// TIA Portal V18 export
VAR_GLOBAL   // PLC tag table "Default tag table"
   "Marca 1" AT %M0.0 : Bool;
   Sumar AT %M0.2 : Bool;
   Entero1 AT %MW2 : Int;
   Restar AT %M0.3 : Bool;
   "Marca 2" AT %M0.1 : Bool;
   Clock_10Hz AT %M100.0 : Bool;
END_VAR
